INTERFACE IGearMover EXTENDS IMover

METHOD Gear : BOOL
VAR_INPUT
	MasterPosition : MC_LREAL;
	SlavePosition : MC_LREAL;
END_VAR
END_METHOD

METHOD inGear : BOOL
VAR_INPUT
END_VAR
END_METHOD

METHOD isMaster : BOOL
VAR_INPUT
END_VAR
END_METHOD

METHOD masterAxis : UDINT
VAR_INPUT
END_VAR
END_METHOD

END_INTERFACE

(* stored: Version 1.1.0.1, ProductVersion 3.1.4024.11
   Itf IGearMover: Id {4e4fd1de-f8b6-49dc-859b-119d358594ce}
   Method Gear: Id {63c7a8e0-32fa-4e3f-84fe-4a57add5caa7}
   Method inGear: Id {e8756b16-d7d4-489b-bbed-8933bde7e4d7}
   Method isMaster: Id {ff5c1c63-a0cf-49dc-80c7-eb87f1062306}
   Method masterAxis: Id {842662f0-2f7b-4c05-82fc-6c80262ae0e0} *)
